Yaskawa INFORM job: Practica meyemberg planos.JBI

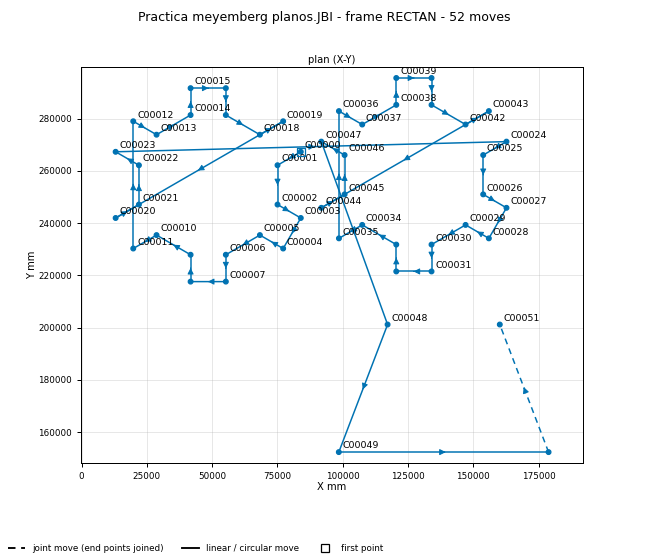
[picture p0: tool path of Practica meyemberg planos.JBI in frame RECTAN, 52 of 52 moves have a stored position in this frame; points joined in program order, loops and branches not executed]
/JOB
//NAME PRACTICA
//POS
///NPOS 7,0,0,0,0,0
///TOOL 0
///POSTYPE RECTAN
///RECTAN
C00000=83958,267331,0,0,0,0
C00001=75045,262185,0,0,0,0
C00002=75045,247127,0,0,0,0
C00003=83958,241981,0,0,0,0
C00004=77208,230290,0,0,0,0
C00005=68295,235435,0,0,0,0
C00006=55254,227906,0,0,0,0
C00007=55254,217615,0,0,0,0
C00008=41754,217614,0,0,0,0
C00009=41754,227906,0,0,0,0
C00010=28713,235435,0,0,0,0
C00011=19800,230290,0,0,0,0
C00012=19800,279022,0,0,0,0
C00013=28713,273877,0,0,0,0
C00014=41754,281406,0,0,0,0
C00015=41754,291698,0,0,0,0
C00016=55254,291698,0,0,0,0
C00017=55254,281406,0,0,0,0
C00018=68295,273877,0,0,0,0
C00019=77208,279022,0,0,0,0
C00020=13050,241981,0,0,0,0
C00021=21963,247127,0,0,0,0
C00022=21963,262185,0,0,0,0
C00023=13050,267331,0,0,0,0
C00024=162726,271227,0,0,0,0
C00025=153813,266081,0,0,0,0
C00026=153813,251022,0,0,0,0
C00027=162726,245876,0,0,0,0
C00028=155976,234185,0,0,0,0
C00029=147063,239331,0,0,0,0
C00030=134022,231802,0,0,0,0
C00031=134022,221510,0,0,0,0
C00032=120522,221510,0,0,0,0
C00033=120522,231802,0,0,0,0
C00034=107481,239331,0,0,0,0
C00035=98568,234185,0,0,0,0
C00036=98568,282918,0,0,0,0
C00037=107481,277772,0,0,0,0
C00038=120522,285302,0,0,0,0
C00039=120522,295593,0,0,0,0
C00040=134022,295593,0,0,0,0
C00041=134022,285302,0,0,0,0
C00042=147063,277772,0,0,0,0
C00043=155976,282918,0,0,0,0
C00044=91818,245876,0,0,0,0
C00045=100731,251022,0,0,0,0
C00046=100731,266081,0,0,0,0
C00047=91818,271227,0,0,0,0
C00048=117197,201182,0,0,0,0
C00049=98516,152325,0,0,0,0
C00050=178844,152325,0,0,0,0
C00051=160163,201182,0,0,0,0
//INST
///DATE 2025/03/24 09:03
///ATTR SC,RW
///GROUP1 RB1
NOP
MOVJ C00000 VJ=25.00
MOVL C00001 V=83.3
MOVL C00002 V=83.3
MOVL C00003 V=83.3
MOVL C00004 V=83.3
MOVL C00005 V=83.3
MOVL C00006 V=83.3
MOVL C00007 V=83.3
MOVL C00008 V=83.3
MOVL C00009 V=83.3
MOVL C00010 V=83.3
MOVL C00011 V=83.3
MOVL C00012 V=83.3
MOVL C00013 V=83.3
MOVL C00014 V=83.3
MOVL C00015 V=83.3
MOVL C00016 V=83.3
MOVL C00017 V=83.3
MOVL C00018 V=83.3
MOVL C00019 V=83.3
MOVL C00020 V=83.3
MOVL C00021 V=83.3
MOVL C00022 V=83.3
MOVL C00023 V=83.3
MOVL C00024 V=83.3
MOVL C00025 V=83.3
MOVL C00026 V=83.3
MOVL C00027 V=83.3
MOVL C00028 V=83.3
MOVL C00029 V=83.3
MOVL C00030 V=83.3
MOVL C00031 V=83.3
MOVL C00032 V=83.3
MOVL C00033 V=83.3
MOVL C00034 V=83.3
MOVL C00035 V=83.3
MOVL C00036 V=83.3
MOVL C00037 V=83.3
MOVL C00038 V=83.3
MOVL C00039 V=83.3
MOVL C00040 V=83.3
MOVL C00041 V=83.3
MOVL C00042 V=83.3
MOVL C00043 V=83.3
MOVL C00044 V=83.3
MOVL C00045 V=83.3
MOVL C00046 V=83.3
MOVL C00047 V=83.3
MOVL C00048 V=83.3
MOVL C00049 V=83.3
MOVL C00050 V=83.3
MOVJ C00051 VJ=25.00
END
